ABB RobotStudio station: FINAL_PROJECT_STATION_HP.rspag

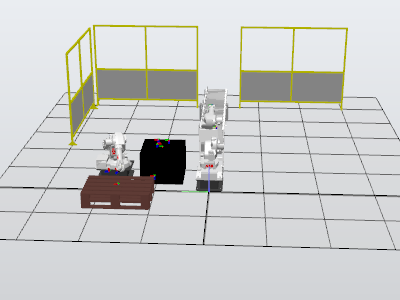
--- station ---
Station FINALPROJECT4 (saved by RobotStudio 23.4.10609.1)
Controller IRB1600_6_120_1, task T_ROB1: task frame (RAPID world) sits at (666.1, 1790.41, 225) mm, rotated rx 0 ry 0 rz -90 deg in the station
Controller IRB1600_6_120, task T_ROB1: task frame (RAPID world) sits at (385, 0, 225) mm in the station
Controller IRB1600_6_120
  mechanical unit ROB_1: IRB1600_6_120__03, 6 joints, base frame (0, 0, 0) mm
Controller IRB1600_6_120_1
  mechanical unit ROB_1: IRB1600_6_120__03_2, 6 joints, base frame (0, 0, 0) mm
Layout (positions relative to the parent item):
  - IRB1600_6_120__03 [mechanism] at (385, 0, 225) mm; joint values [0.0036, 0.1187, -0.2098, -0.0033, 0.8765, 0.0046] (rad or m)
      links: Base, Link1, Link2, Link3, Link4, Link5, Link6
  - Conveyor1 [part] at (1000, -200, 0) mm, size 3033 x 590 x 945 mm
  - VacuumPenToolSC [smart component] at (1234.72, 2.87, 1191.79) mm, rotated rx -180 ry 45 rz -180 deg
      signals: DI diAttacher, DO doAttacher
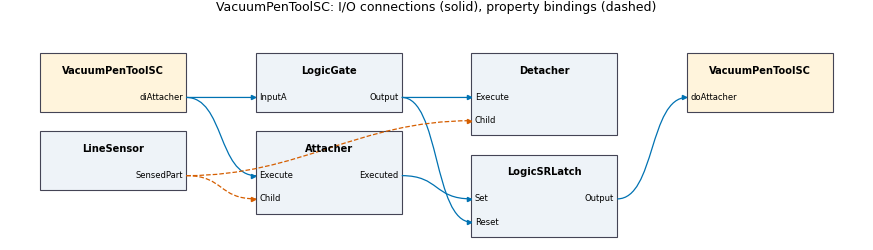
      connections:
        VacuumPenToolSC.diAttacher -> LogicGate.InputA
        LogicGate.Output -> Detacher.Execute
        Attacher.Executed -> LogicSRLatch.Set
        LogicSRLatch.Output -> VacuumPenToolSC.doAttacher
        VacuumPenToolSC.diAttacher -> Attacher.Execute
        LogicGate.Output -> LogicSRLatch.Reset
        LineSensor.SensedPart => Attacher.Child
        LineSensor.SensedPart => Detacher.Child
    - VacuumPenTool [mechanism] at (0, 0, 0) mm
        TCP VacuumTool at (106.34, 126.01, 0.37) mm, rotated rx -90 ry 0 rz -45 deg
        TCP PenTool at (-174.29, 194.28, 0.18) mm, rotated rx -90 ry 0 rz 45 deg
        links: DoubleToolVacuumPencil
    - LineSensor [smart component, from Components\LineSensor.rslib]
        properties: Start=[0.107 -0.00037 0.127]; End=[0.114 0 0.134]; Radius=0.001; SensedPart=(none); SensedPoint=[0 0 0]; Length=0.00990640701768306; Tag=(none)
      - _sensorPart_ [part], size 8.4 x 2.4 x 8.4 mm
    - Attacher [smart component, from Components\Attacher.rslib]
        properties: Parent=VacuumPenTool; Flange=0; Child=(none); Mount=false; Offset=[0 0 0]; Orientation=[0 0 0]
    - Detacher [smart component, from Components\Detacher.rslib]
        properties: Child=(none); KeepPosition=true
    - LogicGate [smart component, from Components\LogicGate.rslib]
        properties: Operator=NOT; Delay=0
    - LogicSRLatch [smart component, from Components\LogicSRLatch.rslib]
  - Robotpedestal1400_H240 [part] at (350, 0, 0) mm, size 660 x 490 x 240 mm
  - Box [part] at (600, 800, 600) mm, size 200 x 200 x 100 mm
  - SmartComponent_1 [smart component]
      signals: DO Sensor, DI PICK, DI StartMotor, DI Pick2, DI Created_box2
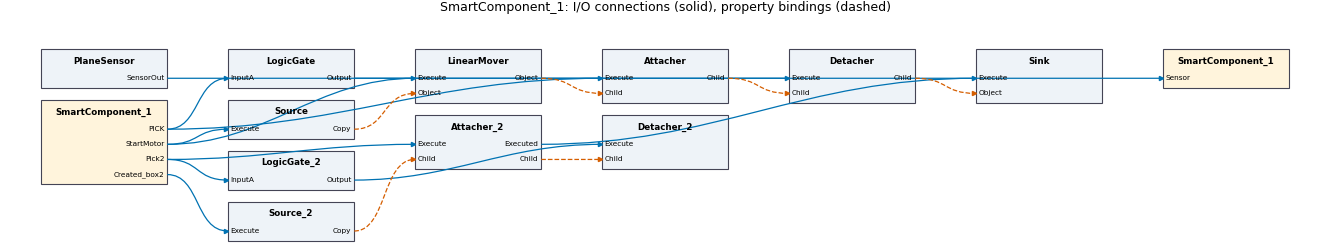
      connections:
        PlaneSensor.SensorOut -> SmartComponent_1.Sensor
        SmartComponent_1.PICK -> Attacher.Execute
        SmartComponent_1.PICK -> LogicGate.InputA
        LogicGate.Output -> Detacher.Execute
        SmartComponent_1.StartMotor -> LinearMover.Execute
        SmartComponent_1.StartMotor -> Source.Execute
        SmartComponent_1.Pick2 -> Attacher_2.Execute
        SmartComponent_1.Pick2 -> LogicGate_2.InputA
        LogicGate_2.Output -> Detacher_2.Execute
        SmartComponent_1.Created_box2 -> Source_2.Execute
        Attacher_2.Executed -> Sink.Execute
        Source.Copy => LinearMover.Object
        LinearMover.Object => Attacher.Child
        Attacher.Child => Detacher.Child
        Attacher_2.Child => Detacher_2.Child
        Source_2.Copy => Attacher_2.Child
        Detacher.Child => Sink.Object
    - LinearMover [smart component, from Components\LinearMover.rslib]
        properties: Object=(none); Direction=[-1 0 0]; Speed=0.4; Reference=Global; ReferenceObject=(none)
    - Source [smart component, from Components\Source.rslib]
        properties: Source=Box; Copy=(none); Parent=(none); Position=[3.750237 -0.0975 0.77206]; Orientation=[0 0 0]; Transient=true; PhysicsBehavior=-1
    - PlaneSensor [smart component, from Components\PlaneSensor.rslib] at (1282.55, -92.67, 747.49) mm
        properties: Origin=[-0.132549993954389 -0.00733450323135224 0.02751387483892]; Axis1=[0 0 0.2]; Axis2=[0 0.2 0]; Tag=(none); SensedPart=(none)
      - _sensorPart_ [part], size 0 x 200 x 200 mm
    - Attacher [smart component, from Components\Attacher.rslib]
        properties: Parent=VacuumPenToolSC; Flange=0; Child=(none); Mount=false; Offset=[0 0 0]; Orientation=[0 0 0]
    - Detacher [smart component, from Components\Detacher.rslib]
        properties: Child=(none); KeepPosition=true
    - LogicGate [smart component, from Components\LogicGate.rslib]
        properties: Operator=NOT; Delay=0
    - Attacher_2 [smart component, from Components\Attacher.rslib]
        properties: Parent=VacuumPenToolSC_2; Flange=0; Child=(none); Mount=false; Offset=[0 0 0]; Orientation=[0 0 0]
    - LogicGate_2 [smart component, from Components\LogicGate.rslib]
        properties: Operator=NOT; Delay=0
    - Detacher_2 [smart component, from Components\Detacher.rslib]
        properties: Child=(none); KeepPosition=true
    - Source_2 [smart component, from Components\Source.rslib]
        properties: Source=Box; Copy=(none); Parent=(none); Position=[0.6 0.8 0.6]; Orientation=[0 0 0]; Transient=true; PhysicsBehavior=-1
    - Sink [smart component, from Components\Sink.rslib]
        properties: Object=(none)
  - WorkTable [part] at (300, 500, 0) mm, size 800 x 800 x 600 mm
  - Robotpedestal1400_H240_2 [part] at (666.1, 1820.41, 0) mm, rotated rx 0 ry 0 rz -90 deg, size 660 x 490 x 240 mm
  - Euro Pallet [graphiccomponentgroup, from Equipment\Euro Pallet.rslib] at (0, 1000, 0) mm, rotated rx 0 ry 0 rz 90 deg
    - Body 1 [part, from Equipment\Euro Pallet.rslib]
  - Euro Pallet_2 [graphiccomponentgroup, from Equipment\Euro Pallet.rslib] at (0, 1000, 140) mm, rotated rx 0 ry 0 rz 90 deg
    - Body 1 [part, from Equipment\Euro Pallet.rslib]
  - Fence_2500 [graphiccomponentgroup, from Equipment\Fence_2500.rslib] at (5000, 500, 0) mm
    - Body 1 [part, from Equipment\Fence_2500.rslib]
    - Body 2 [part, from Equipment\Fence_2500.rslib]
  - IRB1600_6_120__03_2 [mechanism] at (666.1, 1790.41, 225) mm, rotated rx 0 ry 0 rz -90 deg; joint values [0, -0.6386, 0.5446, 0, 0.6068, 3.0556] (rad or m)
      links: Base, Link1, Link2, Link3, Link4, Link5, Link6
  - VacuumPenToolSC_2 [smart component] at (-399.82, 1585.87, 550.62) mm, rotated rx 180 ry -45 rz 90 deg
      signals: DI diAttacher, DO doAttacher
      connections:
        VacuumPenToolSC_2.diAttacher -> LogicGate.InputA
        LogicGate.Output -> Detacher.Execute
        Attacher.Executed -> LogicSRLatch.Set
        LogicSRLatch.Output -> VacuumPenToolSC_2.doAttacher
        VacuumPenToolSC_2.diAttacher -> Attacher.Execute
        LogicGate.Output -> LogicSRLatch.Reset
        LineSensor.SensedPart => Attacher.Child
        LineSensor.SensedPart => Detacher.Child
    - VacuumPenTool [mechanism] at (-835.61, 999.64, -255.78) mm, rotated rx 0 ry 90 rz -180 deg
        TCP VacuumTool at (106.34, 126.01, 0.37) mm, rotated rx -90 ry 0 rz -45 deg
        TCP PenTool at (-174.29, 194.28, 0.18) mm, rotated rx -90 ry 0 rz 45 deg
        links: DoubleToolVacuumPencil
    - LineSensor [smart component, from Components\LineSensor.rslib]
        properties: Start=[0.107 -0.00037 0.127]; End=[0.114 0 0.134]; Radius=0.001; SensedPart=(none); SensedPoint=[0 0 0]; Length=0.00990640701768306; Tag=(none)
      - _sensorPart_ [part], size 8.4 x 2.4 x 8.4 mm
    - Attacher [smart component, from Components\Attacher.rslib]
        properties: Parent=VacuumPenTool; Flange=0; Child=(none); Mount=false; Offset=[0 0 0]; Orientation=[0 0 0]
    - Detacher [smart component, from Components\Detacher.rslib]
        properties: Child=(none); KeepPosition=true
    - LogicGate [smart component, from Components\LogicGate.rslib]
        properties: Operator=NOT; Delay=0
    - LogicSRLatch [smart component, from Components\LogicSRLatch.rslib]
  - Part_1 [part], size 800 x 1200 x 290 mm
  - LogicGate [smart component, from Components\LogicGate.rslib]
      properties: Operator=AND; Delay=0
  - Fence_2500_2 [graphiccomponentgroup, from Equipment\Fence_2500.rslib] at (5000, -3000, 0) mm
    - Body 1 [part, from Equipment\Fence_2500.rslib]
    - Body 2 [part, from Equipment\Fence_2500.rslib]
  - Fence_2500_3 [graphiccomponentgroup, from Equipment\Fence_2500.rslib] at (4700, 3000, 0) mm, rotated rx 0 ry 0 rz 90 deg
    - Body 1 [part, from Equipment\Fence_2500.rslib]
    - Body 2 [part, from Equipment\Fence_2500.rslib]
Attachment: VacuumPenToolSC is attached to IRB1600_6_120__03 / Link6
Attachment: VacuumPenToolSC_2 is attached to IRB1600_6_120__03_2 / Link6
Attachment: VacuumPenTool is attached to IRB1600_6_120__03_2 / Link6
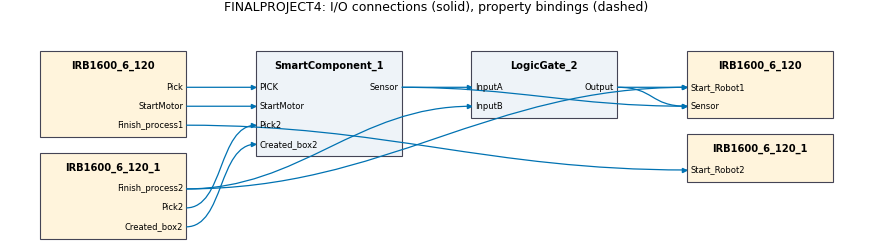
Station logic (signal -> signal, property => property):
  IRB1600_6_120.Pick -> SmartComponent_1.PICK
  IRB1600_6_120.StartMotor -> SmartComponent_1.StartMotor
  IRB1600_6_120.Finish_process1 -> IRB1600_6_120_1.Start_Robot2
  SmartComponent_1.Sensor -> LogicGate_2.InputA
  IRB1600_6_120_1.Finish_process2 -> LogicGate_2.InputB
  LogicGate_2.Output -> IRB1600_6_120.Start_Robot1
  LogicGate_2.Output -> IRB1600_6_120.Sensor
  IRB1600_6_120_1.Finish_process2 -> IRB1600_6_120.Start_Robot1
  SmartComponent_1.Sensor -> IRB1600_6_120.Sensor
  IRB1600_6_120_1.Pick2 -> SmartComponent_1.Pick2
  IRB1600_6_120_1.Created_box2 -> SmartComponent_1.Created_box2

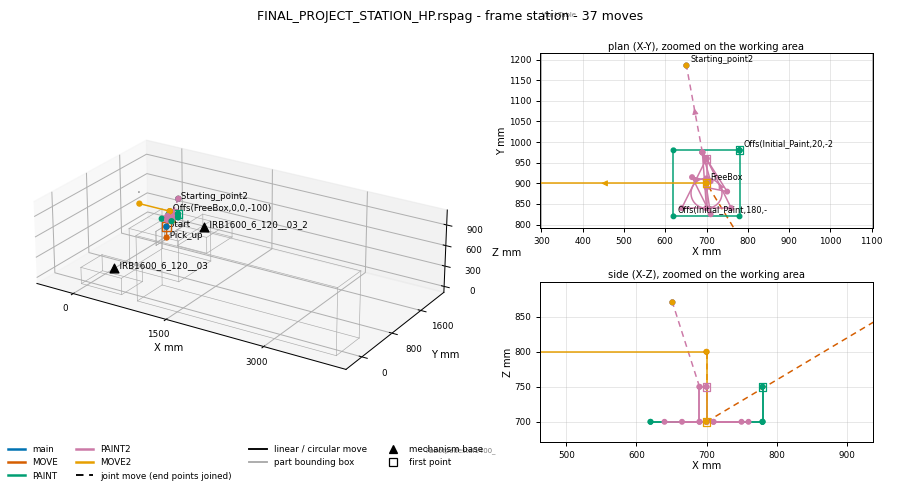
[picture p0: tool path of FINAL_PROJECT_STATION_HP.rspag in frame station, 37 of 39 moves have a stored position in this frame; points joined in program order, loops and branches not executed]
--- Controller Data/IRB1600_6_120/RAPID/TASK1/PROGMOD/CalibData.mod ---
MODULE CalibData
    PERS tooldata VacuumTool:=[TRUE,[[106.338,-0.37,126.015],[0.923879533,0,0.382683432,0]],[1,[0,0,1],[1,0,0,0],0,0,0]];
    PERS tooldata PenTool:=[TRUE,[[-174.289,-0.18,194.277],[0.923879533,0,-0.382683432,0]],[1,[0,0,1],[1,0,0,0],0,0,0]];
    TASK PERS wobjdata WorkBox:=[FALSE,TRUE,"",[[763.637,-97.5,647.06],[0,0,1,0]],[[0,0,0],[1,0,0,0]]];
    TASK PERS wobjdata WorkTable:=[FALSE,TRUE,"",[[315,900,375],[0,0,1,0]],[[0,0,0],[1,0,0,0]]];
    TASK PERS wobjdata WorkPaint_Box:=[FALSE,TRUE,"",[[415,800,475],[0,0,1,0]],[[0,0,0],[1,0,0,0]]];
ENDMODULE

--- Controller Data/IRB1600_6_120/RAPID/TASK1/PROGMOD/Module1.mod ---
MODULE Module1
    CONST robtarget Pinitial:=[[852.772943391,-2.385137119,882.676861768],[0.13052623,0,0.991444856,0],[-1,0,-1,0],[9E+09,9E+09,9E+09,9E+09,9E+09,9E+09]];
    CONST robtarget Ppickup:=[[863.637,2.5,647.06],[0,0,1,0],[0,0,0,0],[9E+09,9E+09,9E+09,9E+09,9E+09,9E+09]];
    CONST robtarget Pfree:=[[315,900,475],[0,0,1,0],[0,0,0,0],[9E+09,9E+09,9E+09,9E+09,9E+09,9E+09]];
    CONST robtarget Start:=[[863.636947578,2.5000019,802.496309732],[-0.000000018,0.000000005,1,0.000000004],[0,-1,0,0],[9E+09,9E+09,9E+09,9E+09,9E+09,9E+09]];
    CONST robtarget Pick_up:=[[-100,100,0],[1,0,0,0],[0,-1,0,0],[9E+09,9E+09,9E+09,9E+09,9E+09,9E+09]];
    CONST robtarget FreeBox:=[[0,0,-100],[1,0,0,0],[0,-1,1,0],[9E+09,9E+09,9E+09,9E+09,9E+09,9E+09]];
    CONST robtarget Initial_Paint:=[[0,200,0],[1,0,0,0],[0,0,0,0],[9E+09,9E+09,9E+09,9E+09,9E+09,9E+09]];

    PROC main()
        SetDO Finish_process1, 0;
        WaitDI Start_Robot1, 1;
        MOVE;
        PAINT;
        MoveJ Start,v1000,fine,VacuumTool\WObj:=wobj0;
        SetDO Finish_process1, 1;
        WaitTime 10;


    ENDPROC
    PROC MOVE()
        MoveJ Start,v1000,fine,VacuumTool\WObj:=wobj0;
        SetDO StartMotor, 1;
        WaitDI Sensor, 1;
        SetDO StartMotor, 0;
        MoveJ Pick_up,v1000,fine,VacuumTool\WObj:=WorkBox;
        SetDO PICK, 1;
        MoveJ Start,v1000,fine,VacuumTool\WObj:=wobj0;
        MoveJ FreeBox,v1000,fine,VacuumTool\WObj:=WorkTable;
        SetDO PICK, 0;
        MoveJ Offs(FreeBox, 0, 0, -100),v1000,fine,VacuumTool\WObj:=WorkTable;
    ENDPROC
    PROC PAINT()
        ! Offsets from: MoveJ Initial_Paint,v1000,fine,PenTool\WObj:=WorkPaint_Box;

        MoveJ Offs(Initial_Paint, 20, -20, -50),v1000,fine,PenTool\WObj:=WorkPaint_Box;
        WaitTime 0.5;
        MoveL Offs(Initial_Paint, 20, -20, 0),v1000,fine,PenTool\WObj:=WorkPaint_Box;
        WaitTime 0.5;
        !SetDO Trace_Robot1, 1;
        MoveL Offs(Initial_Paint, 180, -20, 0),v100,fine,PenTool\WObj:=WorkPaint_Box;
        WaitTime 0.5;
        MoveL Offs(Initial_Paint, 180, -180, 0),v100,fine,PenTool\WObj:=WorkPaint_Box;
        WaitTime 0.5;
        MoveL Offs(Initial_Paint, 20, -180, 0),v100,fine,PenTool\WObj:=WorkPaint_Box;
        WaitTime 0.5;
        MoveL Offs(Initial_Paint, 20, -20, 0),v100,fine,PenTool\WObj:=WorkPaint_Box;
        WaitTime 0.5;
        !SetDO Trace_Robot1, 0;
        MoveL Offs(Initial_Paint, 20, -20, -50),v100,fine,PenTool\WObj:=WorkPaint_Box;

    ENDPROC
ENDMODULE

--- Controller Data/IRB1600_6_120_1/RAPID/TASK1/PROGMOD/CalibData.mod ---
MODULE CalibData
    PERS tooldata VacuumTool:=[TRUE,[[106.338,-0.37,126.015],[0.923879533,0,0.382683432,0]],[1,[0,0,1],[1,0,0,0],0,0,0]];
    PERS tooldata PenTool:=[TRUE,[[-174.289,-0.18,194.277],[0.923879533,0,-0.382683432,0]],[1,[0,0,1],[1,0,0,0],0,0,0]];
    PERS tooldata Tooldata_1:=[TRUE,[[106.338,-0.37,126.015],[0.923879533,0,0.382683432,0]],[1,[0,0,1],[1,0,0,0],0,0,0]];
    PERS tooldata Tooldata_2:=[TRUE,[[-174.289,-0.18,194.277],[0.923879533,0,-0.382683432,0]],[1,[0,0,1],[1,0,0,0],0,0,0]];
    TASK PERS wobjdata WorkDraw_Box:=[FALSE,TRUE,"",[[790.41,-66.099,475],[0,1,0,0]],[[0,0,0],[1,0,0,0]]];
    TASK PERS wobjdata WorkVacuum:=[FALSE,TRUE,"",[[790.41,133.901,475],[0,0,1,0]],[[0,0,0],[1,0,0,0]]];
    TASK PERS wobjdata Workpallet:=[FALSE,TRUE,"",[[790.41,-666.099,65],[0,0,1,0]],[[0,0,0],[1,0,0,0]]];
ENDMODULE

--- Controller Data/IRB1600_6_120_1/RAPID/TASK1/PROGMOD/Module1.mod ---
MODULE Module1
    CONST robtarget Target_10:=[[1086.004966084,-0.180000018,1232.056023362],[0.793353358,0,0.608761406,0],[-1,0,-1,0],[9E+09,9E+09,9E+09,9E+09,9E+09,9E+09]];
    CONST robtarget Starting_point2:=[[604.952418193,-14.791673835,645.639378613],[0.034245553,0.98981165,0.02598571,0.135738289],[0,-1,1,0],[9E+09,9E+09,9E+09,9E+09,9E+09,9E+09]];
    CONST robtarget Start_line:=[[200,0,0],[1,0,0,0],[-1,0,1,0],[9E+09,9E+09,9E+09,9E+09,9E+09,9E+09]];
    CONST robtarget Pick_up2:=[[-100,-100,0],[1,0,0,0],[0,0,0,0],[9E+09,9E+09,9E+09,9E+09,9E+09,9E+09]];
    CONST robtarget FreeBox2:=[[600,-400,0],[1,0,0,0],[-1,0,-2,0],[9E+09,9E+09,9E+09,9E+09,9E+09,9E+09]];
    PERS bool type := TRUE;
    VAR num i :=0;
    VAR num offset_stack :=-100;

    PROC main()
        MoveL Starting_point2,v1000,z100,PenTool\WObj:=wobj0;
        SetDO Finish_process2, 1;
        WaitDI Start_Robot2, 1;
        SetDO Finish_process2, 0;
        PAINT2;
        MOVE2;

    ENDPROC

    PROC PAINT2()
        !MoveL Starting_point2,v1000,z100,PenTool\WObj:=wobj0;
        !MoveL Start_line,v1000,z100,PenTool\WObj:=WorkDraw_Box;
        IF type = FALSE THEN
            MoveL Offs(Start_line,-160,-100,-50),v100,fine,PenTool\WObj:=WorkDraw_Box;
            WaitTime 0.5;
            MoveL Offs(Start_line,-160,-100,0),v100,fine,PenTool\WObj:=WorkDraw_Box;
            WaitTime 0.5;
            !SetDO Trace2, 1;
            MoveL Offs(Start_line,-40,-40,0),v100,fine,PenTool\WObj:=WorkDraw_Box;
            WaitTime 0.5;
            MoveL Offs(Start_line,-40,-160,0),v100,fine,PenTool\WObj:=WorkDraw_Box;
            WaitTime 0.5;
            MoveL Offs(Start_line,-160,-100,0),v100,fine,PenTool\WObj:=WorkDraw_Box;
            WaitTime 0.5;
            MoveL Offs(Start_line,-40,-100,0),v100,fine,PenTool\WObj:=WorkDraw_Box;
            WaitTime 0.5;
            MoveC Offs(Start_line,-78.5,-137.5,0),Offs(Start_line,-112,-100,0),v100,fine,PenTool\WObj:=WorkDraw_Box;
            MoveC Offs(Start_line,-78.5,-62.5,0),Offs(Start_line,-40,-100,0),v100,fine,PenTool\WObj:=WorkDraw_Box;
            WaitTime 0.5;
            !SetDO Trace2, 0;
            MoveL Offs(Start_line,-40,-100,-50),v100,fine,PenTool\WObj:=WorkDraw_Box;

        ELSE
            MoveL Offs(Start_line,-175,-90,-50),v100,fine,PenTool\WObj:=WorkDraw_Box;
            WaitTime 0.5;
            MoveL Offs(Start_line,-175,-90,0),v100,fine,PenTool\WObj:=WorkDraw_Box;
            WaitTime 0.5;
            !SetDO Trace2, 1;
            MoveL Offs(Start_line,-80,-150,0),v100,fine,PenTool\WObj:=WorkDraw_Box;
            WaitTime 0.5;
            MoveL Offs(Start_line,-90,-100,0),v100,fine,PenTool\WObj:=WorkDraw_Box;
            WaitTime 0.5;
            MoveL Offs(Start_line,-25,-110,0),v100,fine,PenTool\WObj:=WorkDraw_Box;
            WaitTime 0.5;
            MoveL Offs(Start_line,-115,-65,0),v100,fine,PenTool\WObj:=WorkDraw_Box;
            WaitTime 0.5;
            MoveL Offs(Start_line,-105,-110,0),v100,fine,PenTool\WObj:=WorkDraw_Box;
            WaitTime 0.5;
            MoveL Offs(Start_line,-175,-90,0),v100,fine,PenTool\WObj:=WorkDraw_Box;
            WaitTime 0.5;
            !SetDO Trace2, 0;
            MoveL Offs(Start_line,-175,-90,-50),v100,fine,PenTool\WObj:=WorkDraw_Box;
            WaitTime 0.5;
            MoveJ Starting_point2,v1000,z100,PenTool\WObj:=wobj0;
        ENDIF


    ENDPROC


    PROC MOVE2()
        SetDO Created_box2, 1;
        MoveJ Pick_up2,v100,fine,VacuumTool\WObj:=WorkVacuum;
        SetDO Pick2, 1;
        MoveL Offs(Pick_up2, 0, 0, -100),v100,fine,VacuumTool\WObj:=WorkVacuum;
        MoveL Offs(Pick_up2, 0, -500, -100),v1000,fine,VacuumTool\WObj:=WorkVacuum;
        IF type = TRUE THEN

            MoveL Offs(FreeBox2,-400,0,offset_stack),v1000,fine,VacuumTool\WObj:=Workpallet;

        ELSE

            MoveL Offs(FreeBox2,-100,0,offset_stack),v1000,fine,VacuumTool\WObj:=Workpallet;
            offset_stack := offset_stack - 100;

        ENDIF


        IF type = TRUE THEN
            type := FALSE;
        ELSE
            type := TRUE;
        ENDIF
        SetDO Pick2, 0;
        SetDO Created_box2, 0;
        MoveL Starting_point2,v1000,z100,PenTool\WObj:=wobj0;
    ENDPROC
ENDMODULE

--- Controller Data/IRB1600_6_120/SYSPAR/EIO.cfg ---
EIO:CFG_1.0:6:1::
#
EIO_SIGNAL:

      -Name "Sensor" -SignalType "DI"

      -Name "StartMotor" -SignalType "DO"

      -Name "Pick" -SignalType "DO"

      -Name "Finish_process1" -SignalType "DO"\
      -Label "Finishes the process of the robot 1"

      -Name "Start_Robot1" -SignalType "DI"

--- Controller Data/IRB1600_6_120_1/SYSPAR/EIO.cfg ---
EIO:CFG_1.0:6:1::
#
EIO_SIGNAL:

      -Name "Start_Robot2" -SignalType "DI"\
      -Label "Digital Input to call the robot2 and start working"

      -Name "Finish_process2" -SignalType "DO"

      -Name "Pick2" -SignalType "DO"

      -Name "Created_box2" -SignalType "DO"
